TYPE ST_valToAccess :
STRUCT
  	severity: BYTE;
	errorSummary:	T_MaxString;
	errorMessage: T_MaxString;
	remediationMessage: T_MaxString;
	telegramSending: STRING(1);
	hmiErrorShow: STRING(1);
END_STRUCT
END_TYPE

(* stored: Version 1.1.0.1, ProductVersion 3.1.4024.12
   DUT ST_valToAccess: Id {df14c275-fac4-4d19-8d12-6472aff80f66} *)
